# EPICS autosave request: softGlueApp/Db/MagCmp_settings.req
$(P)$(H)MagCmp-$(N)_SAMPLE_Signal
$(P)$(H)MagCmp-$(N)_AGTB_Signal
$(P)$(H)MagCmp-$(N)_ANEB_Signal

$(P)$(H)MagCmp-$(N)_BDIR_Signal
$(P)$(H)MagCmp-$(N)_BCK_Signal
